RoboDK station: New P2_MobileRobot.rdk

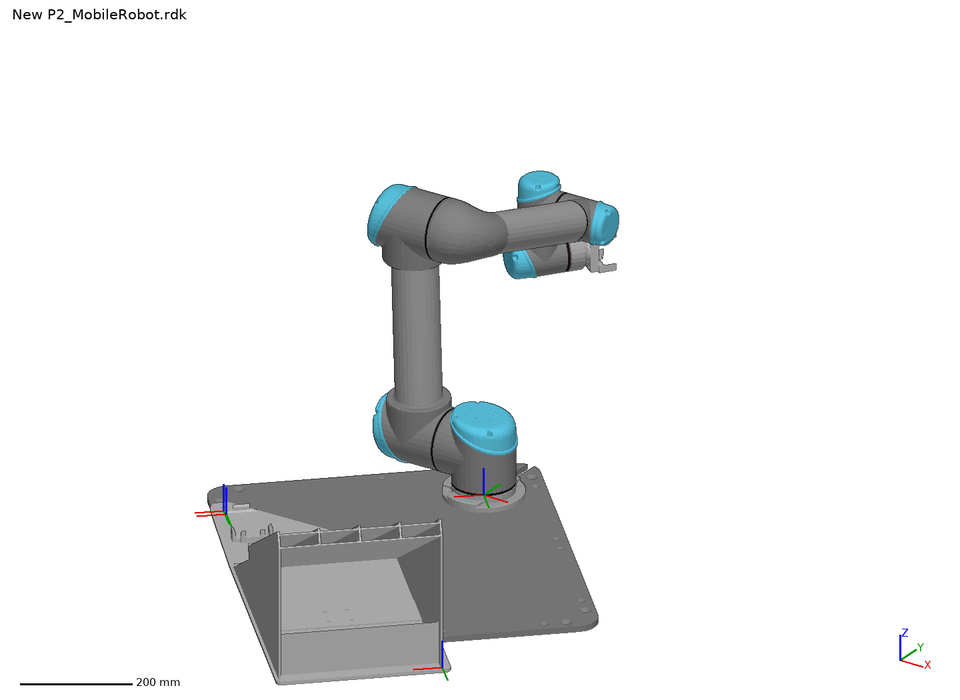
[picture v0: the station drawn from its stored meshes, robots at their saved joint values, targets as dots, program paths as lines]
Station New P2_MobileRobot (saved by RoboDK 5.6.8). Poses are relative to the parent item; angles as X-Y-Z fixed-axis rotations.
  - frame UR5 Base at (0, 0, 0) mm
    - robot UR5: 6 axes
        modified DH rows (alpha deg, a mm, theta deg, d mm): 0, 0, 0, 89.2; 90, 0, 180, 0; 0, 425, 0, 0; 0, 392, 0, 109.3; -90, 0, 0, 94.75; 90, 0, 180, 82.5
        joint limits [-360, -360, -360, -360, -360, -360] to [360, 360, 360, 360, 360, 360]; home [0, -90, -90, 0, 90, 0]; saved at [-87.43, -92.62, 110.29, -17.67, 126.9, -90]
      - tool Tool 1, TCP at (0, 0, 0) mm, rotated rx 0 ry 0 rz 180 deg
        - object Gripper FINAL at (-668.04, -188.63, 987) mm, size 106.1 x 65 x 52 mm, geometry from Gripper FINAL.stl
    - frame Rotated Base at (0, 0, 0) mm, rotated rx 0 ry 0 rz -135 deg
      - object Platform at (185, -115, -10) mm, rotated rx 90 ry 0 rz 90 deg, size 670 x 10.5 x 600 mm, geometry from Phone assembly solution.step
      - frame Plate - Frame at (466, -15, 0) mm
        - object Plate at (20, 569.5, 0) mm, rotated rx 0 ry 0 rz 180 deg, size 315 x 736.3 x 6 mm, geometry from BoltPlade_v0 (3).stl
        - frame Mounting station at (0, 25, 6) mm
          - object Mounting station V5 at (9, 57.5, 10.5) mm, rotated rx 90 ry 0 rz -90 deg, size 125 x 25 x 72 mm, geometry from Mounting station V5.stl
          - frame Frame 5 at (-270, 680, 0) mm
            - object Phone_thing_Andre_happy (1) at (-416.1, -483.4, 115.27) mm, size 295 x 466.8 x 287.1 mm, geometry from Phone_thing_Andre_happy (1).stl
  - Python program Prog1 (listed below)

--- Python program Prog1 ---
# Type help("robodk.robolink") or help("robodk.robomath") for more information
# Press F5 to run the script
# Documentation: https://robodk.com/doc/en/RoboDK-API.html
# Reference:     https://robodk.com/doc/en/PythonAPI/robodk.html
# Note: It is not required to keep a copy of this file, your Python script is saved with your RDK project

# You can also use the new version of the API:
from robodk import robolink    # RoboDK API
from robodk import robomath    # Robot toolbox
RDK = robolink.Robolink()

# Forward and backwards compatible use of the RoboDK API:
# Remove these 2 lines to follow python programming guidelines
from robodk import *      # RoboDK API
from robolink import *    # Robot toolbox
# Link to RoboDK
# RDK = Robolink()

# Notify user:
print('To edit this program:\nright click on the Python program, then, select "Edit Python script"')

# Program example:
item = RDK.Item('base')
if item.Valid():
    print('Item selected: ' + item.Name())
    print('Item posistion: ' + repr(item.Pose()))

print('Items in the station:')
itemlist = RDK.ItemList()
print(itemlist)

# Provoking an exception will display the console output if you run this script from RoboDK
raise Exception('Program not edited.')
